{attribute 'GeneratedUsingTerminal: EP2316-0008-0017'}
{attribute addProperty BoxType "EP2316-0008-0017"}
{attribute addProperty Id "AdsAddrAT %I*AMSADDR8StateAT %I*UINT2"}
{attribute addProperty CRC "854291690"}
{attribute addProperty Size "10"}
TYPE InfoData_32EB74EA :
STRUCT
	{attribute addProperty Name "AdsAddr"}
	AdsAddr AT %I* : AMSADDR;
	{attribute addProperty Name "State"}
	State AT %I* : UINT;
END_STRUCT
END_TYPE

(* stored: Version 1.2.0.0, ProductVersion 3.1.4024.9
   DUT InfoData_32EB74EA: Id {79ce1a8d-27d2-4ee3-8811-0a28d8273c2c} *)
